PROGRAM MAIN
VAR
    _app : AppContext;
END_VAR

_app.Run();
_app.RtcSynchronize(true, '', 60);

END_PROGRAM

(* stored: Version 1.1.0.1, ProductVersion 3.1.4024.12
   POU MAIN: Id {f73432eb-0afd-4ae9-a59a-cc056bccad50}, SpecialFunc None *)
